FUNCTION_BLOCK FB_SaMElementSuspended EXTENDS FB_SaMElement
VAR
END_VAR

END_FUNCTION_BLOCK

(* stored: Version 1.1.0.1
   POU FB_SaMElementSuspended: Id {6cb875bc-0af2-08e2-33e8-85b12bc09e51}, SpecialFunc None *)
